// SIMATIC S7-200 SMART project (STEP 7-Micro/WIN SMART), CPU SR40

SYMBOL_TABLE System Symbols
Always_On        SM0.0    // Always ON
First_Scan_On    SM0.1    // ON for the first scan cycle only
Clock_1s         SM0.5    // Clock pulse that is ON for 0.5 s, OFF for 0.5 s, for a duty cycle time of 1 s.
END_SYMBOL_TABLE

ORGANIZATION_BLOCK MAIN:OB1
TITLE=Program Comments
BEGIN
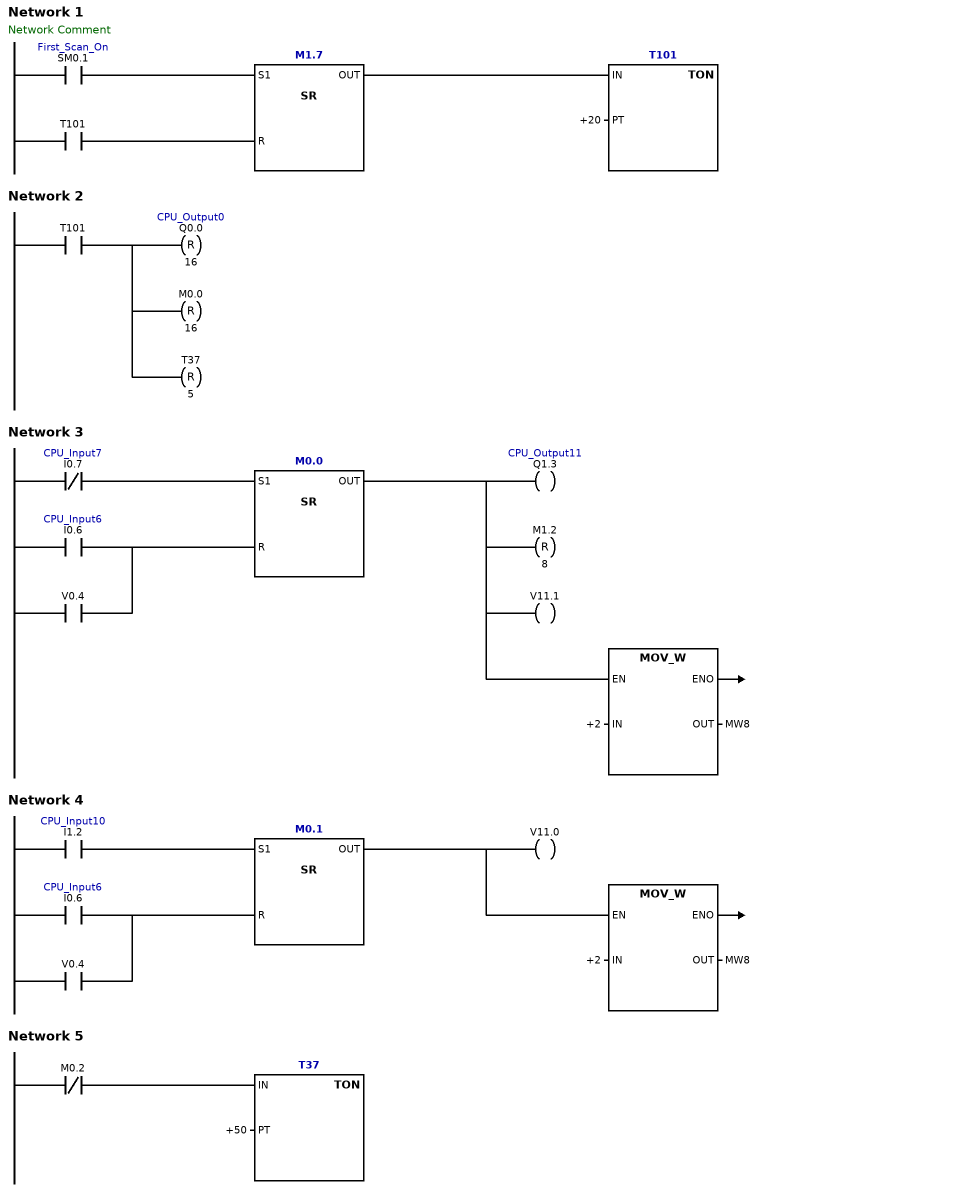
Network 1
// Network Comment
LD     First_Scan_On:SM0.1
LD     T101
NOT
A      M1.7
OLD
=      M1.7
TON    T101, +20
Network 2
LD     T101
R      CPU_Output0:Q0.0, 16
R      M0.0, 16
R      T37, 5
Network 3
LDN    CPU_Input7:I0.7
LD     CPU_Input6:I0.6
O      V0.4
NOT
A      M0.0
OLD
=      M0.0
=      CPU_Output11:Q1.3
R      M1.2, 8
=      V11.1
MOVW   +2, MW8
Network 4
LD     CPU_Input10:I1.2
LD     CPU_Input6:I0.6
O      V0.4
NOT
A      M0.1
OLD
=      M0.1
=      V11.0
MOVW   +2, MW8
Network 5
LDN    M0.2
TON    T37, +50
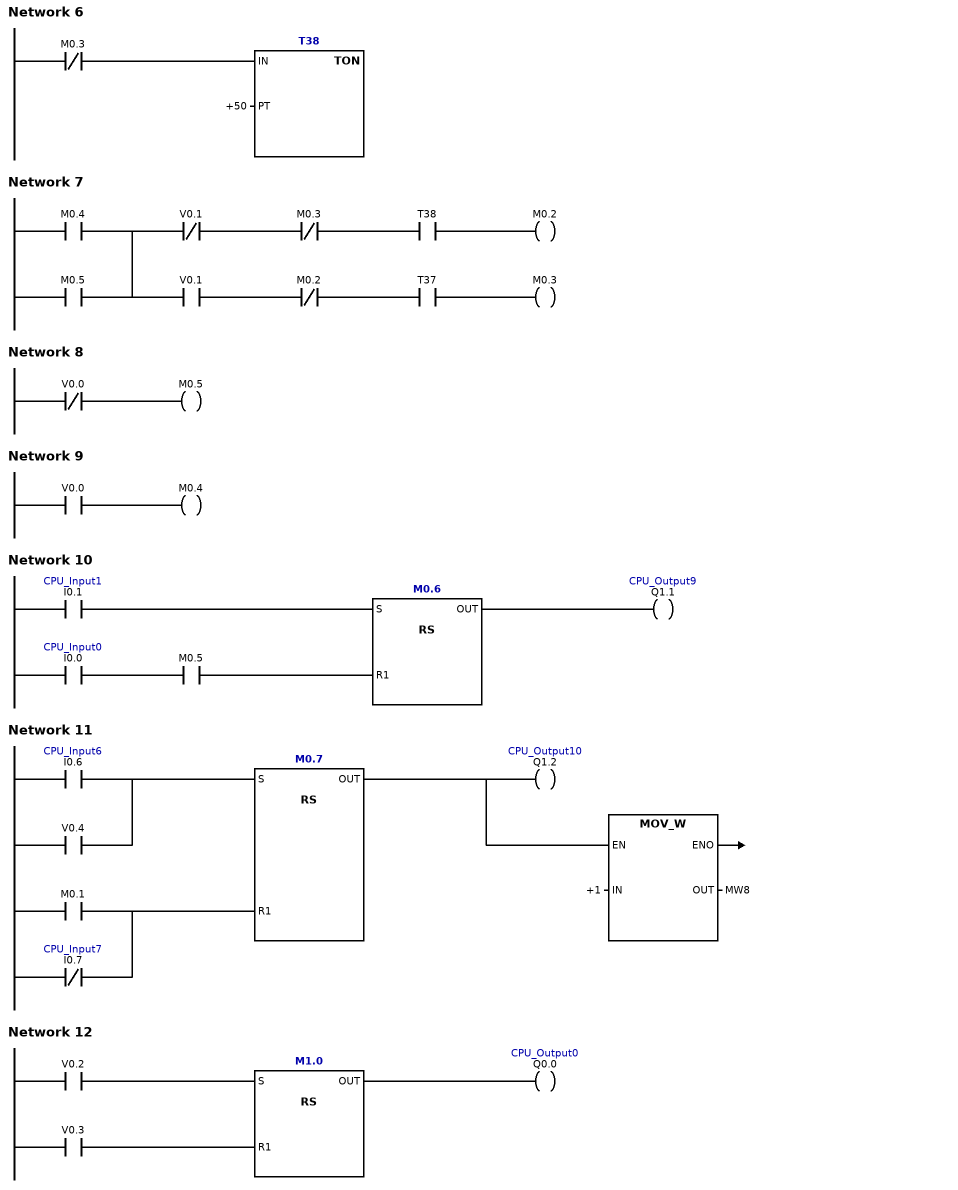
Network 6
LDN    M0.3
TON    T38, +50
Network 7
LD     M0.4
O      M0.5
LPS
AN     V0.1
AN     M0.3
A      T38
=      M0.2
LPP
A      V0.1
AN     M0.2
A      T37
=      M0.3
Network 8
LDN    V0.0
=      M0.5
Network 9
LD     V0.0
=      M0.4
Network 10
LD     CPU_Input1:I0.1
LD     CPU_Input0:I0.0
A      M0.5
NOT
LPS
A      M0.6
=      M0.6
LPP
ALD
O      M0.6
=      M0.6
=      CPU_Output9:Q1.1
Network 11
LD     CPU_Input6:I0.6
O      V0.4
LD     M0.1
ON     CPU_Input7:I0.7
NOT
LPS
A      M0.7
=      M0.7
LPP
ALD
O      M0.7
=      M0.7
=      CPU_Output10:Q1.2
MOVW   +1, MW8
Network 12
LD     V0.2
LD     V0.3
NOT
LPS
A      M1.0
=      M1.0
LPP
ALD
O      M1.0
=      M1.0
=      CPU_Output0:Q0.0
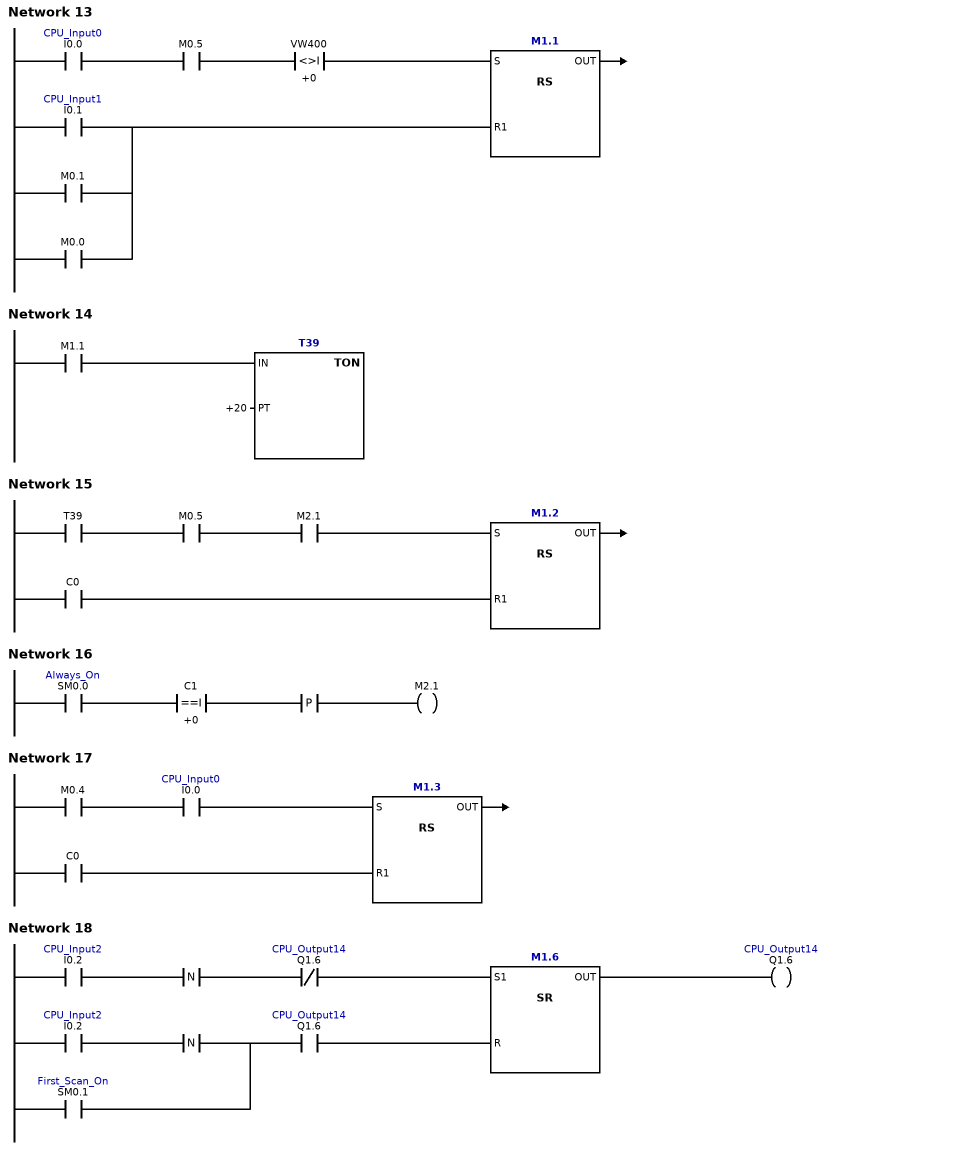
Network 13
LD     CPU_Input0:I0.0
A      M0.5
AW<>   VW400, +0
LD     CPU_Input1:I0.1
O      M0.1
O      M0.0
NOT
LPS
A      M1.1
=      M1.1
LPP
ALD
O      M1.1
=      M1.1
Network 14
LD     M1.1
TON    T39, +20
Network 15
LD     T39
A      M0.5
A      M2.1
LD     C0
NOT
LPS
A      M1.2
=      M1.2
LPP
ALD
O      M1.2
=      M1.2
Network 16
LD     Always_On:SM0.0
AW=    C1, +0
EU
=      M2.1
Network 17
LD     M0.4
A      CPU_Input0:I0.0
LD     C0
NOT
LPS
A      M1.3
=      M1.3
LPP
ALD
O      M1.3
=      M1.3
Network 18
LD     CPU_Input2:I0.2
ED
AN     CPU_Output14:Q1.6
LD     CPU_Input2:I0.2
ED
O      First_Scan_On:SM0.1
A      CPU_Output14:Q1.6
NOT
A      M1.6
OLD
=      M1.6
=      CPU_Output14:Q1.6
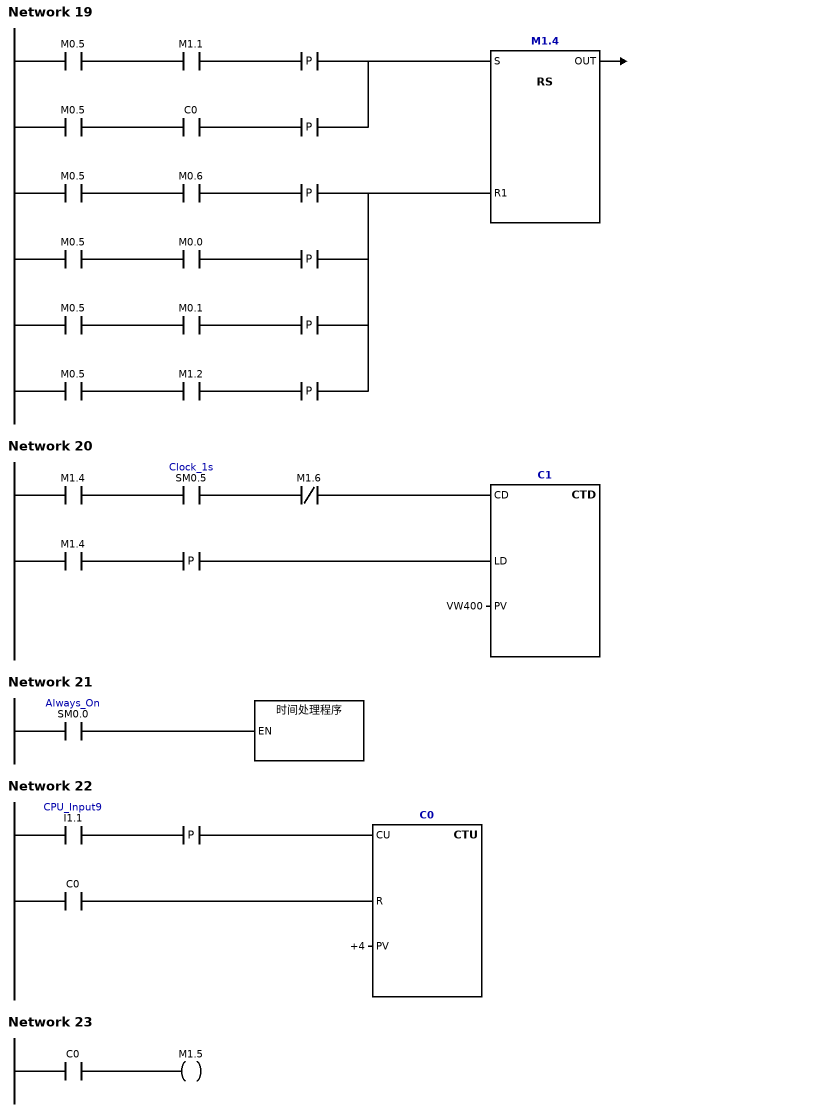
Network 19
LD     M0.5
A      M1.1
EU
LD     M0.5
A      C0
EU
OLD
LD     M0.5
A      M0.6
EU
LD     M0.5
A      M0.0
EU
OLD
LD     M0.5
A      M0.1
EU
OLD
LD     M0.5
A      M1.2
EU
OLD
NOT
LPS
A      M1.4
=      M1.4
LPP
ALD
O      M1.4
=      M1.4
Network 20
LD     M1.4
A      Clock_1s:SM0.5
AN     M1.6
LD     M1.4
EU
CTD    C1, VW400
Network 21
LD     Always_On:SM0.0
CALL   时间处理程序:SBR1
Network 22
LD     CPU_Input9:I1.1
EU
LD     C0
CTU    C0, +4
Network 23
LD     C0
=      M1.5
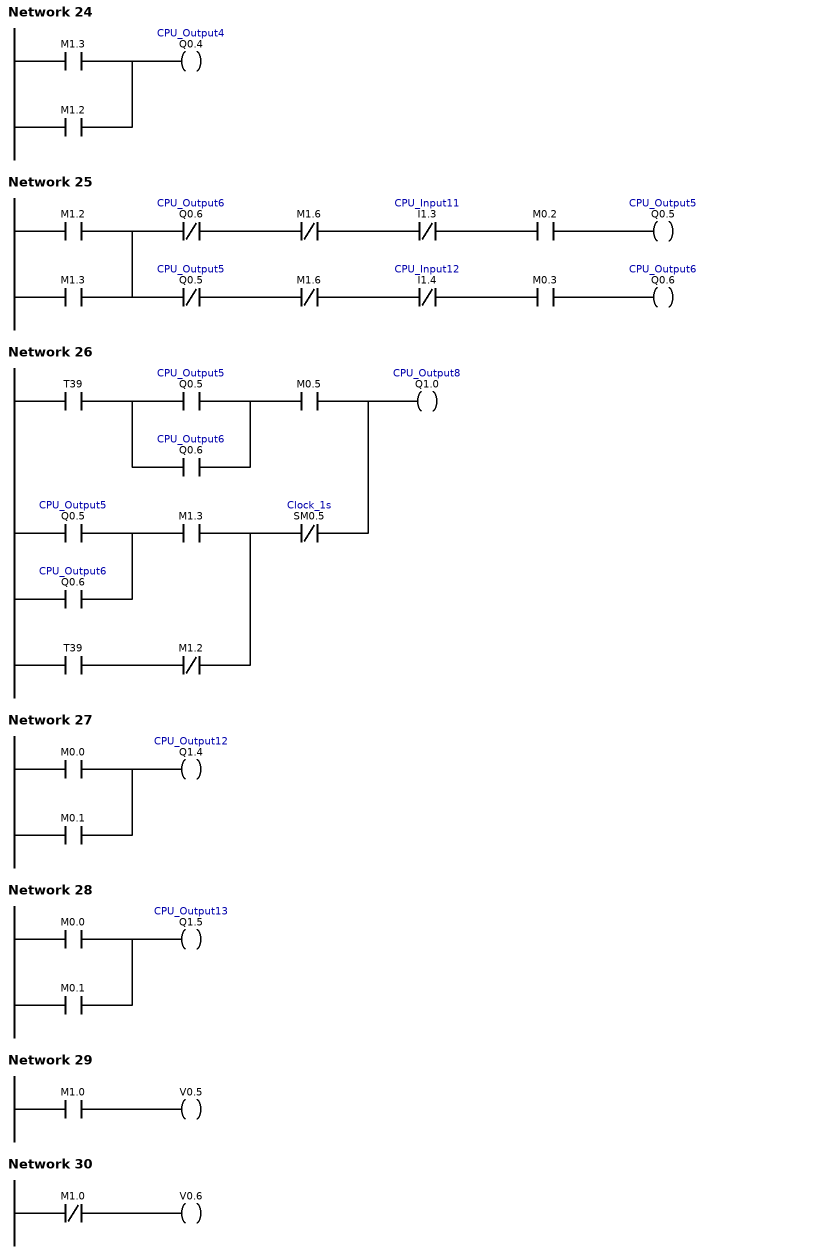
Network 24
LD     M1.3
O      M1.2
=      CPU_Output4:Q0.4
Network 25
LD     M1.2
O      M1.3
LPS
AN     CPU_Output6:Q0.6
AN     M1.6
AN     CPU_Input11:I1.3
A      M0.2
=      CPU_Output5:Q0.5
LPP
AN     CPU_Output5:Q0.5
AN     M1.6
AN     CPU_Input12:I1.4
A      M0.3
=      CPU_Output6:Q0.6
Network 26
LD     T39
LD     CPU_Output5:Q0.5
O      CPU_Output6:Q0.6
ALD
A      M0.5
LD     CPU_Output5:Q0.5
O      CPU_Output6:Q0.6
A      M1.3
LD     T39
AN     M1.2
OLD
AN     Clock_1s:SM0.5
OLD
=      CPU_Output8:Q1.0
Network 27
LD     M0.0
O      M0.1
=      CPU_Output12:Q1.4
Network 28
LD     M0.0
O      M0.1
=      CPU_Output13:Q1.5
Network 29
LD     M1.0
=      V0.5
Network 30
LDN    M1.0
=      V0.6
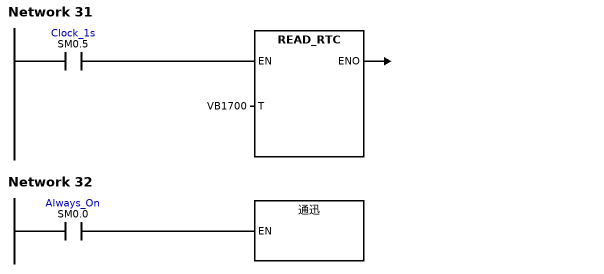
Network 31
LD     Clock_1s:SM0.5
TODR   VB1700
Network 32
LD     Always_On:SM0.0
CALL   通迅:SBR0
END_ORGANIZATION_BLOCK

SUBROUTINE_BLOCK 通迅:SBR0
TITLE=Subroutine Comments
BEGIN
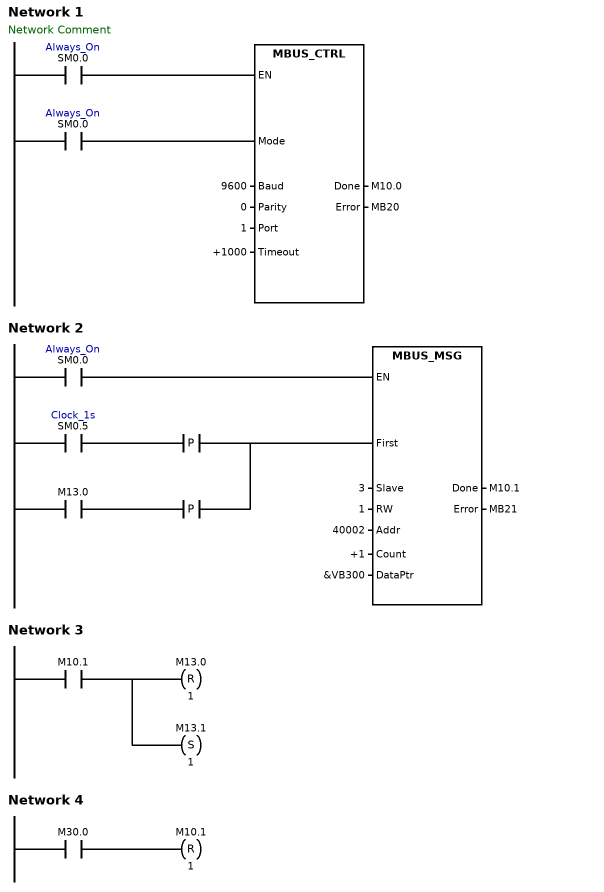
Network 1
// Network Comment
LD     Always_On:SM0.0
=      L60.0
LD     Always_On:SM0.0
=      L63.7
LD     L60.0
CALL   MBUS_CTRL:SBR2, L63.7, 9600, 0, 1, +1000, M10.0, MB20
Network 2
LD     Always_On:SM0.0
=      L60.0
LD     Clock_1s:SM0.5
EU
LD     M13.0
EU
OLD
=      L63.7
LD     L60.0
CALL   MBUS_MSG:SBR3, L63.7, 3, 1, 40002, +1, &VB300, M10.1, MB21
Network 3
LD     M10.1
R      M13.0, 1
S      M13.1, 1
Network 4
LD     M30.0
R      M10.1, 1
END_SUBROUTINE_BLOCK

SUBROUTINE_BLOCK 时间处理程序:SBR1
TITLE=
BEGIN
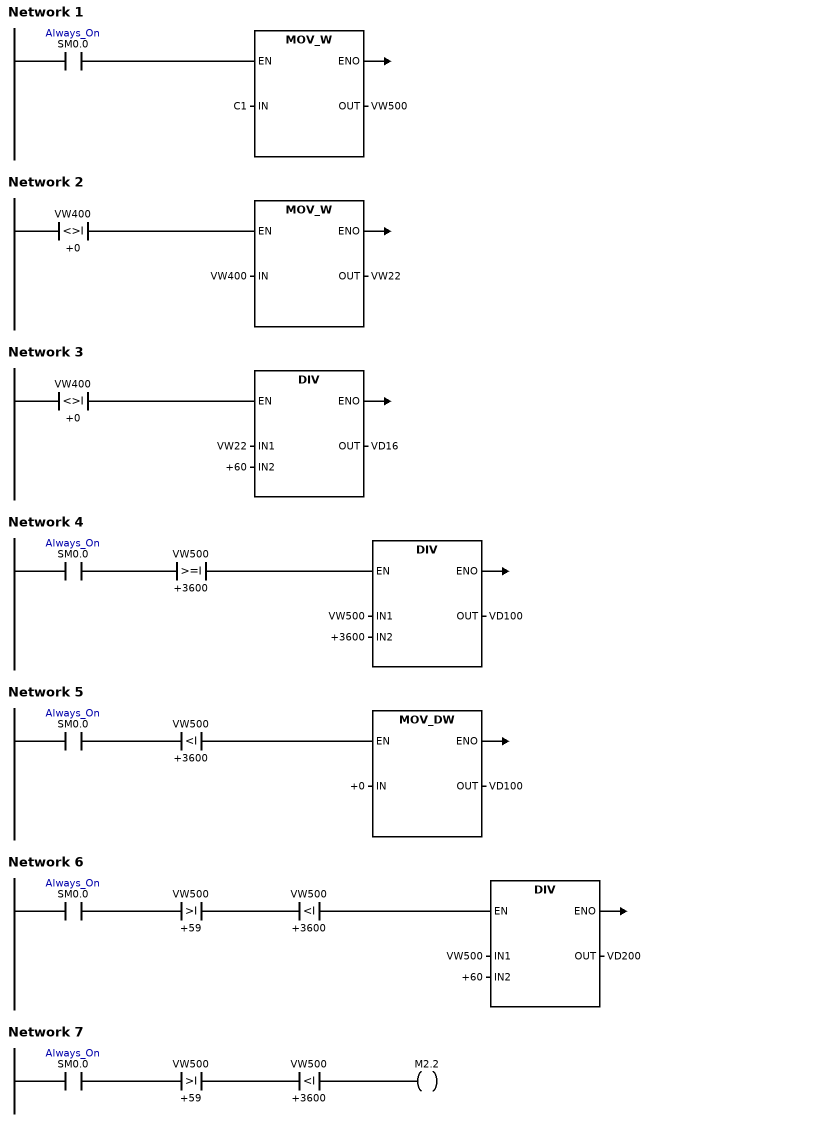
Network 1
LD     Always_On:SM0.0
MOVW   C1, VW500
Network 2
LDW<>  VW400, +0
MOVW   VW400, VW22
Network 3
LDW<>  VW400, +0
MOVW   VW22, VW18
DIV    +60, VD16
Network 4
LD     Always_On:SM0.0
AW>=   VW500, +3600
MOVW   VW500, VW102
DIV    +3600, VD100
Network 5
LD     Always_On:SM0.0
AW<    VW500, +3600
MOVD   +0, VD100
Network 6
LD     Always_On:SM0.0
AW>    VW500, +59
AW<    VW500, +3600
MOVW   VW500, VW202
DIV    +60, VD200
Network 7
LD     Always_On:SM0.0
AW>    VW500, +59
AW<    VW500, +3600
=      M2.2
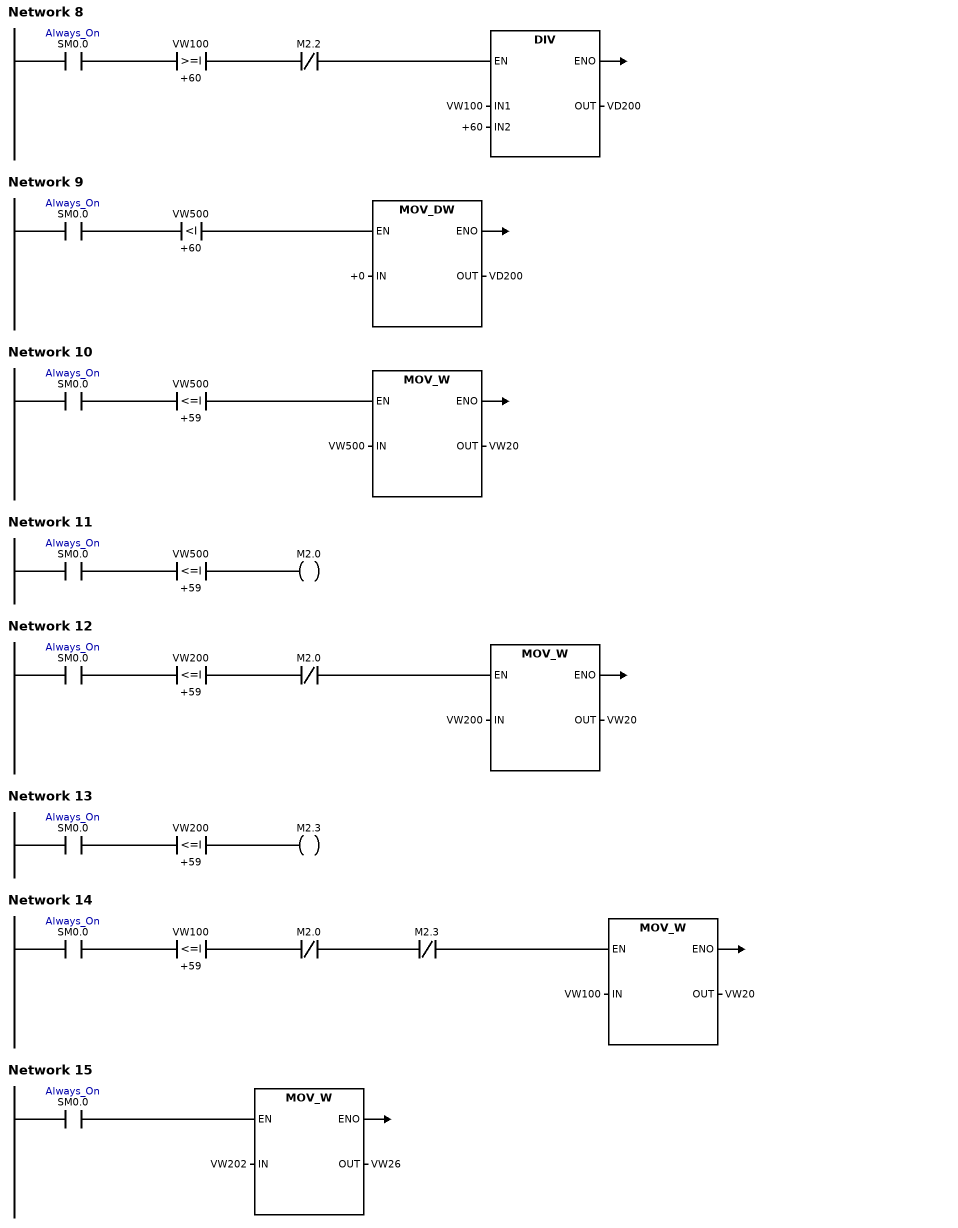
Network 8
LD     Always_On:SM0.0
AW>=   VW100, +60
AN     M2.2
MOVW   VW100, VW202
DIV    +60, VD200
Network 9
LD     Always_On:SM0.0
AW<    VW500, +60
MOVD   +0, VD200
Network 10
LD     Always_On:SM0.0
AW<=   VW500, +59
MOVW   VW500, VW20
Network 11
LD     Always_On:SM0.0
AW<=   VW500, +59
=      M2.0
Network 12
LD     Always_On:SM0.0
AW<=   VW200, +59
AN     M2.0
MOVW   VW200, VW20
Network 13
LD     Always_On:SM0.0
AW<=   VW200, +59
=      M2.3
Network 14
LD     Always_On:SM0.0
AW<=   VW100, +59
AN     M2.0
AN     M2.3
MOVW   VW100, VW20
Network 15
LD     Always_On:SM0.0
MOVW   VW202, VW26
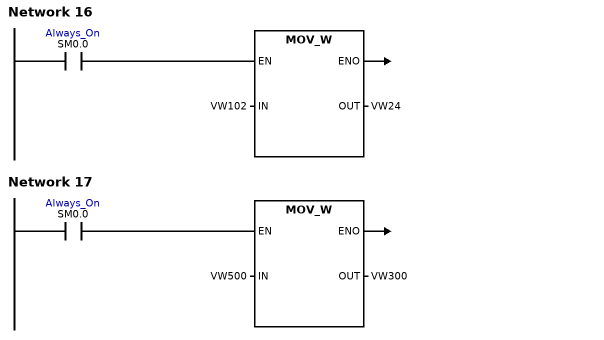
Network 16
LD     Always_On:SM0.0
MOVW   VW102, VW24
Network 17
LD     Always_On:SM0.0
MOVW   VW500, VW300
END_SUBROUTINE_BLOCK

// SBR2: protected block, not included

// SBR3: protected block, not included

// SBR4: protected block, not included

// INT1: protected block, not included
